Staubli VAL3: start.pgx

program start()
begin
  call test_ventouse()
end
